(*
SPDX-FileCopyrightText: Â© 2026 Oleksandr Tiutyk <trofimich@gmail.com>
SPDX-License-Identifier: MIT
License: https://opensource.org/license/mit
*)

(*!
<summary>Digital input automation component supporting normally-open and normally-closed contacts.</summary>
<description>
Reads raw hardware inputs during the automation input processing phase and tracks edge changes.
</description>
*)

FUNCTION_BLOCK DigitalInput EXTENDS TOF_Automation.InputLeafAutomationComponent
	IMPLEMENTS IDigitalInput, TOF_Core.IIOBindable
VAR_STAT
	{attribute 'hide'} 
	_ClassName : STRING := __POUNAME();
END_VAR
VAR
	{attribute 'hide'} 
	_ContactType : CONTACT_TYPE;
	
	_CurrentValue : BOOL;
	_PreviousValue : BOOL;
	
	_RawValue : REFERENCE TO BOOL;
END_VAR

(*!
<summary>Binds component to a raw boolean process image variable.</summary>
<param name="rawValue">Reference to physical boolean input variable.</param>
*)
METHOD BindToIO
VAR_INPUT
	rawValue : REFERENCE TO BOOL;
END_VAR
_RawValue REF= rawValue;
END_METHOD

(*!
<summary>Gets whether the component is bound to a valid physical IO variable.</summary>
*)
{attribute 'monitoring' := 'call'}
PROPERTY FINAL BoundToIO : BOOL
GET
BoundToIO := __ISVALIDREF(_RawValue);
END_GET
END_PROPERTY

(*!
<summary>Indicates whether the logical Value has changed compared to the previous cycle.</summary>
*)
{attribute 'monitoring' := 'call'}
PROPERTY FINAL Changed : BOOL
GET
Changed := _CurrentValue <> _PreviousValue;
END_GET
END_PROPERTY

(*!
<summary>Gets the class name of the component.</summary>
*)
{attribute 'monitoring' := 'call'}
PROPERTY ClassName : REFERENCE TO STRING
GET
ClassName REF= _ClassName;
END_GET
END_PROPERTY

(*!
<summary>Gets or sets electrical contact configuration.</summary>
*)
{attribute 'monitoring' := 'call'}
PROPERTY FINAL ContactType : CONTACT_TYPE
GET
ContactType := _ContactType;
END_GET
SET
_ContactType := ContactType;
END_SET
END_PROPERTY

(*!
<summary>Gets the namespace name of the component.</summary>
*)
{attribute 'monitoring' := 'call'}
PROPERTY NamespaceName : REFERENCE TO STRING
GET
NamespaceName REF= CurrentNamespace.Name;
END_GET
END_PROPERTY

(*!
<summary>Evaluates current input value according to contact type configuration.</summary>
*)
METHOD PROTECTED OnProcessInput
_PreviousValue := _CurrentValue;

IF __ISVALIDREF(_RawValue) THEN
	IF _ContactType = CONTACT_TYPE.NORMALLY_CLOSED THEN
		_CurrentValue := NOT _RawValue;
	ELSE
		_CurrentValue := _RawValue;
	END_IF
END_IF
END_METHOD

(*!
<summary>Gets the memory size of the instance.</summary>
*)
{attribute 'monitoring' := 'call'}
PROPERTY SelfSize : ULINT
GET
SelfSize := XSIZEOF(THIS^);
END_GET
END_PROPERTY

(*!
<summary>Gets evaluated logical boolean state of the input.</summary>
*)
{attribute 'monitoring' := 'call'}
{attribute 'OPC.UA.DA' := '1'}
{attribute 'OPC.UA.DA.Access' := '1'}
PROPERTY FINAL Value : BOOL
GET
Value := _CurrentValue;
END_GET
END_PROPERTY

END_FUNCTION_BLOCK

(* stored: Version 1.1.0.1
   POU DigitalInput: Id {c6d1eaf1-9cc8-4dbf-a584-1b04597f0f65}, SpecialFunc None
   Folder Overriden methods: Id {914655df-4424-4133-ac94-26668b3cec6e}
   Method BindToIO: Id {655d2c7c-c530-408b-863c-1bfa26ef7b01}
   Property BoundToIO: Id {56a705c1-66d1-44d2-91fe-eff8dee2a4c4}
   Get Get: Id {0bc6dabb-05f8-4f35-8118-477b477e120f}
   Property Changed: Id {25fa1762-2c5f-4829-a6e8-7bee560cce1e}
   Get Get: Id {7ff589e4-c33f-4f73-855a-49a7e43cb387}
   Property ClassName: Id {e5420b88-e83e-4617-b101-8fff6688087b}
   Get Get: Id {6468f6c3-92d1-4468-8b70-32b585af0c9f}
   Property ContactType: Id {4b3ab9a4-1fa8-4610-aac4-3d8f85976c52}
   Get Get: Id {4c06f3af-47f7-4db5-9cef-e5f746e7fe2d}
   Set Set: Id {6875e153-f614-4371-a701-9a573e1339ec}
   Property NamespaceName: Id {51db961c-fcae-40ea-a673-1cae49d16d4c}
   Get Get: Id {59a6fc02-c8b3-4706-a9f3-a476bd008abe}
   Method OnProcessInput: Id {a28fb2bd-177b-4c2a-9df6-5bfe86d8083d}
   Property SelfSize: Id {3cc9639a-e2ec-49ce-8c2d-d08927803438}
   Get Get: Id {cad1d82f-8f76-41da-8b67-afbeb31a8e85}
   Property Value: Id {435debbb-bc61-4a95-9bd6-b412ba0f938a}
   Get Get: Id {5d93ee31-a76c-4b10-880a-8a0871008a6c} *)
